FUNCTION_BLOCK AxisResetTestSuite 
VAR
	StubAxis : AXIS_REF;
	iStubTask : I_Task;
	TestAxisReset : CoEResetTask := (AxisRef := StubAxis);
	ObjTestSuite : TestSuite<TestSuiteParameter.MaxTestCount>(ResultFile := JUnitResultFile) := (TestSuiteName := 'Object Test Suite');
END_VAR

DoesAcceptExecute_Test();
DoesTaskAbortClearBusy_Test();
DoesTaskAccept_Test();
RejectResetWhileResetting_Test();

METHOD DoesAcceptExecute_Test : BOOL
VAR_INST
	Expected : HRESULT;
	Actual	 : HRESULT;
END_VAR
IF ObjTestSuite.Test(__POUNAME()).ExecuteTest() THEN
	Expected := s_OK;
	Actual := TestAxisReset.Reset();
	TestAxisReset.Abort();
	ObjTestSuite.Test(__POUNAME()).AssertEqual(Expected, Actual);
END_IF
END_METHOD

METHOD DoesTaskAbortClearBusy_Test
VAR_INST
	Expected : BOOL := FALSE;
	Actual	 : BOOL;
END_VAR
IF ObjTestSuite.Test(__POUNAME()).ExecuteTest() THEN
	TestAxisReset.Reset();
	TestAxisReset.Abort();
	Actual := TestAxisReset.Busy;
	ObjTestSuite.Test(__POUNAME()).AssertEqual(Expected, Actual);
END_IF
END_METHOD

METHOD DoesTaskAccept_Test
VAR_INST
	Expected : BOOL := TRUE;
	Actual	 : bool;
END_VAR
IF ObjTestSuite.Test(__POUNAME()).ExecuteTest() THEN
	Actual := SUCCEEDED(TestAxisReset.Reset());
	TestAxisReset.Abort();
	ObjTestSuite.Test(__POUNAME()).AssertEqual(Expected, Actual);
END_IF
END_METHOD

METHOD RejectResetWhileResetting_Test : BOOL
VAR_INST
	Expected : BOOL := TRUE;
	Actual	 : BOOL;
END_VAR
IF ObjTestSuite.Test(__POUNAME()).ExecuteTest() THEN
	TestAxisReset.Reset();
	Actual := FAILED(TestAxisReset.Reset());
	ObjTestSuite.Test(__POUNAME()).AssertEqual(Expected, Actual);
END_IF
END_METHOD

END_FUNCTION_BLOCK

(* stored: Version 1.1.0.1
   POU AxisResetTestSuite: Id {35388208-47d1-43d3-9073-bac1bf114263}, SpecialFunc None
   Method DoesAcceptExecute_Test: Id {08513cf5-caba-4c77-9c71-3b8a7a80c814}
   Method DoesTaskAbortClearBusy_Test: Id {b4acbce4-731b-4329-9277-0416ac626e31}
   Method DoesTaskAccept_Test: Id {215a4d80-e8c0-4f6d-808b-dc5958b3620f}
   Method RejectResetWhileResetting_Test: Id {0b718029-0f95-45b5-9686-fbc342e36ff7} *)
